# EPICS substitutions: AD{{ cookiecutter.driver_name }}/iocs/{{ cookiecutter.driver_name }}IOC/iocBoot/ioc{{ cookiecutter.driver_name }}/auto_settings.req
file "AD{{ cookiecutter.driver_name }}_settings.req",  P=$(P),  R=cam1:
file "NDStdArrays_settings.req",  P=$(P),  R=image1:
file "commonPlugin_settings.req", P=$(P)
